FUNCTION_BLOCK fb_prod_rate_ctrl

VAR_INPUT
	kc: REAL;
	ti:REAL;
	ts:REAL;
	hi:REAL;
	lo:REAL;
	x0:REAL := 0;
	set_prod_rate: REAL := g_set_production;
	//xmv17: REAL;

END_VAR

VAR_OUTPUT
	Prodsp: REAL;
	Fp: REAL;
END_VAR

VAR
	
	slewrate_limiter: fb_slewrate_limiter := (pos_slewrate_limit := 0.286875, neg_slewrate_limit := -0.286875);
	prodsp_scaled: REAL;
	prodrate_discrete_pi: fb_discrete_pi := (kc := 3.2, ti := 120, ts := g_Ts_base, hi := 30, lo := -30, x0:=0);
END_VAR

VAR CONSTANT
	ProdspGain: REAL := 100/22.89;
END_VAR

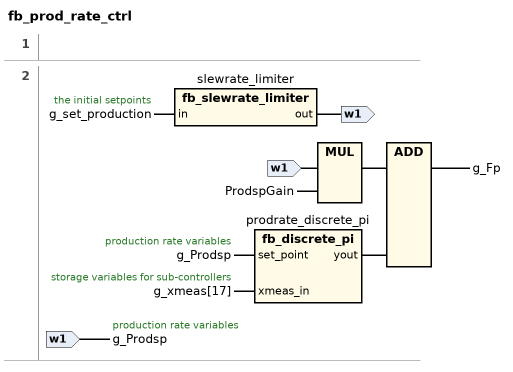
// NETWORK 1

// NETWORK 2
//   g_set_production: the initial setpoints
//   g_Prodsp: production rate variables
//   g_xmeas[17]: storage variables for sub-controllers
slewrate_limiter(in := g_set_production); // fb_slewrate_limiter
prodrate_discrete_pi(set_point := g_Prodsp, xmeas_in := g_xmeas[17]); // fb_discrete_pi
g_Fp := slewrate_limiter.out * ProdspGain + prodrate_discrete_pi.yout;
g_Prodsp := slewrate_limiter.out;

END_FUNCTION_BLOCK

(* stored: Version 1.1.0.1, ProductVersion 3.1.0.26
   POU fb_prod_rate_ctrl: Id {12afc640-1cc9-456e-b128-0a54a95b7ca0} *)
